screen "Configuraciones_3" 800x480, template "Template_3"
   IOField "I/O field_1" at 51,95 size 96x32; FormatPattern s99999
      ProcessValue <- "UDT_Objetos_Bombas_BC-11_frecuencia"
   TextField "Text field_1" at 75,36 size 32x20; Text 'XXX'
   TextField "Text field_3" at 60,57 size 74x36; Text 'Frecuencia Trabajo'
   IOField "I/O field_3" at 49,241 size 96x32; FormatPattern 999
      ProcessValue <- "UDT_Objetos_Sensores_Especiales_COT-01_operacion_bajo"
   TextField "Text field_4" at 71,180 size 32x20; Text 'XXX'
   TextField "Text field_5" at 40,202 size 114x36; Text 'Rango operación bajo'
   IOField "I/O field_4" at 49,314 size 96x32; FormatPattern 999
      ProcessValue <- "UDT_Objetos_Sensores_Especiales_COT-01_operacion_alto"
   TextField "Text field_6" at 40,275 size 114x36; Text 'Rango operación alto'
   IOField "I/O field_5" at 49,387 size 96x32; FormatPattern 999
      ProcessValue <- "UDT_Objetos_Sensores_Especiales_COT-01_trabajo_alto"
   TextField "Text field_7" at 63,348 size 67x36; Text 'Punto de trabajo'
   IOField "I/O field_6" at 201,240 size 96x32; FormatPattern 9999
      ProcessValue <- "UDT_Objetos_Flujo_FI-11_operacion_alto"
   TextField "Text field_8" at 295,179 size 38x20; Text 'FI-11'
   TextField "Text field_9" at 192,201 size 114x36; Text 'Rango operación bajo'
   IOField "I/O field_7" at 201,313 size 96x32; FormatPattern 9999
      ProcessValue <- "UDT_Objetos_Flujo_FI-11_operacion_alto"
   TextField "Text field_10" at 192,274 size 114x36; Text 'Rango operación alto'
   IOField "I/O field_8" at 201,386 size 96x32; FormatPattern 9999
      ProcessValue <- "UDT_Objetos_Flujo_FI-11_trabajo_alto"
   TextField "Text field_11" at 208,347 size 82x36; Text 'Punto de trabajo alto'
   IOField "I/O field_9" at 331,240 size 96x32; FormatPattern 9999
      ProcessValue <- "UDT_Objetos_Flujo_FI-11_trabajo_bajo"
   TextField "Text field_12" at 338,201 size 85x36; Text 'Punto de trabajo bajo'
   IOField "I/O field_2" at 484,240 size 96x32; FormatPattern s9999
      ProcessValue <- "UDT_Objetos_Flujo_FI-09_operacion_bajo"
   TextField "Text field_2" at 572,179 size 32x20; Text 'XXX'
   TextField "Text field_13" at 475,201 size 114x36; Text 'Rango operación bajo'
   IOField "I/O field_10" at 484,313 size 96x32; FormatPattern s9999
      ProcessValue <- "UDT_Objetos_Flujo_FI-09_operacion_alto"
   TextField "Text field_14" at 475,274 size 114x36; Text 'Rango operación alto'
   IOField "I/O field_11" at 484,386 size 96x32; FormatPattern s9999
      ProcessValue <- "UDT_Objetos_Flujo_FI-09_trabajo_alto"
   TextField "Text field_15" at 491,347 size 82x36; Text 'Punto de trabajo alto'
   IOField "I/O field_12" at 614,240 size 96x32; FormatPattern s9999
      ProcessValue <- "UDT_Objetos_Flujo_FI-09_trabajo_bajo"
   TextField "Text field_16" at 621,201 size 85x36; Text 'Punto de trabajo bajo'
   Button "Template_Button_7" at 0,440 size 99x39; TextOff 'COT'; PictureOff "Left_Arrow"
      on Click: ActivateScreen("Configuraciones_2", 0)
   Button "Template_Button_8" at 700,441 size 99x39; TextOff 'PT'; PictureOff "Right_Arrow"
      on Click: ActivateScreen("Configuraciones_4", 0)

screen "Configuraciones_4" 800x480, template "Template_3"
   IOField "I/O field_1" at 51,95 size 96x32; FormatPattern s99999
      ProcessValue <- "UDT_Objetos_Bombas_BC-11_frecuencia"
   TextField "Text field_1" at 75,36 size 32x20; Text 'XXX'
   TextField "Text field_3" at 60,57 size 74x36; Text 'Frecuencia Trabajo'
   IOField "I/O field_3" at 49,241 size 96x32; FormatPattern 999
      ProcessValue <- "UDT_Objetos_Sensores_Especiales_COT-01_operacion_bajo"
   TextField "Text field_4" at 71,180 size 32x20; Text 'XXX'
   TextField "Text field_5" at 40,202 size 114x36; Text 'Rango operación bajo'
   IOField "I/O field_4" at 49,314 size 96x32; FormatPattern 999
      ProcessValue <- "UDT_Objetos_Sensores_Especiales_COT-01_operacion_alto"
   TextField "Text field_6" at 40,275 size 114x36; Text 'Rango operación alto'
   IOField "I/O field_5" at 49,387 size 96x32; FormatPattern 999
      ProcessValue <- "UDT_Objetos_Sensores_Especiales_COT-01_trabajo_alto"
   TextField "Text field_7" at 63,348 size 67x36; Text 'Punto de trabajo'
   IOField "I/O field_6" at 201,240 size 96x32; FormatPattern 9999
      ProcessValue <- "UDT_Objetos_Flujo_FI-08_operacion_bajo"
   TextField "Text field_8" at 295,179 size 38x20; Text 'FI-08'
   TextField "Text field_9" at 192,201 size 114x36; Text 'Rango operación bajo'
   IOField "I/O field_7" at 201,313 size 96x32; FormatPattern 9999
      ProcessValue <- "UDT_Objetos_Flujo_FI-08_operacion_alto"
   TextField "Text field_10" at 192,274 size 114x36; Text 'Rango operación alto'
   IOField "I/O field_8" at 201,386 size 96x32; FormatPattern 9999
      ProcessValue <- "UDT_Objetos_Flujo_FI-08_trabajo_alto"
   TextField "Text field_11" at 208,347 size 82x36; Text 'Punto de trabajo alto'
   IOField "I/O field_9" at 331,240 size 96x32; FormatPattern 9999
      ProcessValue <- "UDT_Objetos_Flujo_FI-08_trabajo_bajo"
   TextField "Text field_12" at 338,201 size 85x36; Text 'Punto de trabajo bajo'
   IOField "I/O field_2" at 484,240 size 96x32; FormatPattern s9999
      ProcessValue <- "UDT_Objetos_Flujo_FI-09_operacion_bajo"
   TextField "Text field_2" at 572,179 size 38x20; Text 'FI-09'
   TextField "Text field_13" at 475,201 size 114x36; Text 'Rango operación bajo'
   IOField "I/O field_10" at 484,313 size 96x32; FormatPattern s9999
      ProcessValue <- "UDT_Objetos_Flujo_FI-09_operacion_alto"
   TextField "Text field_14" at 475,274 size 114x36; Text 'Rango operación alto'
   IOField "I/O field_11" at 484,386 size 96x32; FormatPattern s9999
      ProcessValue <- "UDT_Objetos_Flujo_FI-09_trabajo_alto"
   TextField "Text field_15" at 491,347 size 82x36; Text 'Punto de trabajo alto'
   IOField "I/O field_12" at 614,240 size 96x32; FormatPattern s9999
      ProcessValue <- "UDT_Objetos_Flujo_FI-09_trabajo_bajo"
   TextField "Text field_16" at 621,201 size 85x36; Text 'Punto de trabajo bajo'
   Button "Template_Button_7" at 0,440 size 99x39; TextOff 'COT'; PictureOff "Left_Arrow"
      on Click: ActivateScreen("Configuraciones_3", 0)
   Button "Template_Button_8" at 700,441 size 99x39; TextOff 'PT'; PictureOff "Right_Arrow"
      on Click: ActivateScreen("Configuraciones_5", 0)

screen "Configuraciones_5" 800x480, template "Template_3"
   IOField "I/O field_6" at 80,88 size 96x32; FormatPattern 9999; Unit  m
      ProcessValue <- "UDT_Objetos_Nivel_RAD-04_rango_alto"
   TextField "Text field_8" at 101,22 size 55x20; Text 'RAD-04'
   TextField "Text field_9" at 71,44 size 114x36; Text 'Rango operacion alto'
   IOField "I/O field_7" at 80,157 size 96x32; FormatPattern 9999; Unit  m
      ProcessValue <- "UDT_Objetos_Nivel_RAD-04_rango_bajo"
   TextField "Text field_10" at 95,129 size 67x20; Text 'Nivel bajo'
   IOField "I/O field_8" at 80,242 size 96x32; FormatPattern 9999; Unit  m
      ProcessValue <- "UDT_Objetos_Nivel_RAD-04_rango_medio_bajo"
   TextField "Text field_11" at 90,198 size 77x36; Text 'Nivel medio bajo'
   IOField "I/O field_9" at 80,327 size 96x32; FormatPattern 9999; Unit  m
      ProcessValue <- "UDT_Objetos_Nivel_RAD-04_rango_medio_alto"
   TextField "Text field_12" at 90,283 size 77x36; Text 'Nivel medio alto'
   IOField "I/O field_1" at 80,397 size 96x32; FormatPattern 9999; Unit  m
      ProcessValue <- "UDT_Objetos_Nivel_RAD-04_rango_alto"
   TextField "Text field_1" at 96,368 size 64x20; Text 'Nivel alto'
   IOField "I/O field_11" at 617,87 size 96x32; FormatPattern 9999; Unit  m
      ProcessValue <- "UDT_Objetos_Nivel_RAD-06_rango_alto"
   TextField "Text field_13" at 638,21 size 55x20; Text 'RAD-06'
   TextField "Text field_14" at 608,43 size 114x36; Text 'Rango operacion alto'
   IOField "I/O field_12" at 617,156 size 96x32; FormatPattern 9999; Unit  m
      ProcessValue <- "UDT_Objetos_Nivel_RAD-06_rango_bajo"
   TextField "Text field_15" at 632,128 size 67x20; Text 'Nivel bajo'
   IOField "I/O field_13" at 617,241 size 96x32; FormatPattern 9999; Unit  m
      ProcessValue <- "UDT_Objetos_Nivel_RAD-06_rango_medio_bajo"
   TextField "Text field_16" at 627,197 size 77x36; Text 'Nivel medio bajo'
   IOField "I/O field_14" at 617,326 size 96x32; FormatPattern 9999; Unit  m
      ProcessValue <- "UDT_Objetos_Nivel_RAD-06_rango_medio_alto"
   TextField "Text field_17" at 627,282 size 77x36; Text 'Nivel medio alto'
   IOField "I/O field_15" at 617,396 size 96x32; FormatPattern 9999; Unit  m
      ProcessValue <- "UDT_Objetos_Nivel_RAD-06_rango_alto(1)"
   TextField "Text field_18" at 633,367 size 64x20; Text 'Nivel alto'
   IOField "I/O field_2" at 350,88 size 96x32; FormatPattern 9999; Unit  m
      ProcessValue <- "UDT_Objetos_Nivel_RAD-05_rango_alto"
   TextField "Text field_2" at 371,22 size 55x20; Text 'RAD-05'
   TextField "Text field_3" at 341,44 size 114x36; Text 'Rango operacion alto'
   IOField "I/O field_3" at 350,157 size 96x32; FormatPattern 9999; Unit  m
      ProcessValue <- "UDT_Objetos_Nivel_RAD-05_rango_bajo"
   TextField "Text field_4" at 365,129 size 67x20; Text 'Nivel bajo'
   IOField "I/O field_4" at 350,242 size 96x32; FormatPattern 9999; Unit  m
      ProcessValue <- "UDT_Objetos_Nivel_RAD-05_rango_medio_bajo"
   TextField "Text field_5" at 360,198 size 77x36; Text 'Nivel medio bajo'
   IOField "I/O field_5" at 350,327 size 96x32; FormatPattern 9999; Unit  m
      ProcessValue <- "UDT_Objetos_Nivel_RAD-05_rango_medio_alto"
   TextField "Text field_6" at 360,283 size 77x36; Text 'Nivel medio alto'
   IOField "I/O field_10" at 350,397 size 96x32; FormatPattern 9999; Unit  m
      ProcessValue <- "UDT_Objetos_Nivel_RAD-05_rango_alto"
   TextField "Text field_7" at 366,368 size 64x20; Text 'Nivel alto'
   Button "Template_Button_7" at 0,440 size 99x39; TextOff 'COT'; PictureOff "Left_Arrow"
      on Click: ActivateScreen("Configuraciones_4", 0)
   Button "Template_Button_8" at 700,441 size 99x39; TextOff 'PT'; PictureOff "Right_Arrow"
      on Click: ActivateScreen("Presion", 0)

screen "Presion" 800x480, template "Template_3"
   IOField "I/O field_6" at 20,87 size 96x32; FormatPattern 9999; Unit  Bar
      ProcessValue <- "UDT_Objetos_Presion_PT-05_operacion_bajo"
   TextField "Text field_8" at 114,26 size 42x20; Text 'PT-05'
   TextField "Text field_9" at 11,48 size 114x36; Text 'Rango operación bajo'
   IOField "I/O field_7" at 20,160 size 96x32; FormatPattern 9999; Unit  Bar
      ProcessValue <- "UDT_Objetos_Presion_PT-05_operacion_alto"
   TextField "Text field_10" at 11,121 size 114x36; Text 'Rango operación alto'
   IOField "I/O field_8" at 149,160 size 96x32; FormatPattern 9999; Unit  Bar
      ProcessValue <- "UDT_Objetos_Presion_PT-05_trabajo_alto"
   TextField "Text field_11" at 156,121 size 82x36; Text 'Punto de trabajo alto'
   IOField "I/O field_9" at 150,87 size 96x32; FormatPattern 9999; Unit  Bar
      ProcessValue <- "UDT_Objetos_Presion_PT-05_trabajo_bajo"
   TextField "Text field_12" at 157,48 size 85x36; Text 'Punto de trabajo bajo'
   Group "Group" at 5,16 size 259x198
   IOField "I/O field_13" at 20,295 size 96x32; FormatPattern 9999; Unit  Bar
      ProcessValue <- "UDT_Objetos_Presion_PT-09_operacion_bajo"
   TextField "Text field_16" at 114,234 size 42x20; Text 'PT-09'
   TextField "Text field_17" at 11,256 size 114x36; Text 'Rango operación bajo'
   IOField "I/O field_14" at 20,368 size 96x32; FormatPattern 9999; Unit  Bar
      ProcessValue <- "UDT_Objetos_Presion_PT-09_operacion_alto"
   TextField "Text field_18" at 11,329 size 114x36; Text 'Rango operación alto'
   IOField "I/O field_15" at 149,368 size 96x32; FormatPattern 9999; Unit  Bar
      ProcessValue <- "UDT_Objetos_Presion_PT-09_trabajo_alto"
   TextField "Text field_19" at 156,329 size 82x36; Text 'Punto de trabajo alto'
   IOField "I/O field_16" at 150,295 size 96x32; FormatPattern 9999; Unit  Bar
      ProcessValue <- "UDT_Objetos_Presion_PT-09_trabajo_bajo"
   TextField "Text field_20" at 157,256 size 85x36; Text 'Punto de trabajo bajo'
   IOField "I/O field_17" at 286,295 size 96x32; FormatPattern 9999; Unit  Bar
      ProcessValue <- "UDT_Objetos_Presion_PT-10_operacion_bajo"
   TextField "Text field_21" at 380,234 size 42x20; Text 'PT-10'
   TextField "Text field_22" at 277,256 size 114x36; Text 'Rango operación bajo'
   IOField "I/O field_18" at 286,368 size 96x32; FormatPattern 9999; Unit  Bar
      ProcessValue <- "UDT_Objetos_Presion_PT-10_operacion_alto"
   TextField "Text field_23" at 277,329 size 114x36; Text 'Rango operación alto'
   IOField "I/O field_19" at 415,368 size 96x32; FormatPattern 9999; Unit  Bar
      ProcessValue <- "UDT_Objetos_Presion_PT-10_trabajo_alto"
   TextField "Text field_24" at 422,329 size 82x36; Text 'Punto de trabajo alto'
   IOField "I/O field_20" at 416,295 size 96x32; FormatPattern 9999; Unit  Bar
      ProcessValue <- "UDT_Objetos_Presion_PT-10_trabajo_bajo"
   TextField "Text field_25" at 423,256 size 85x36; Text 'Punto de trabajo bajo'
   IOField "I/O field_21" at 553,295 size 96x32; FormatPattern 9999; Unit  Bar
      ProcessValue <- "UDT_Objetos_Presion_PT-11_operacion_bajo"
   TextField "Text field_26" at 647,234 size 42x20; Text 'PT-11'
   TextField "Text field_27" at 544,256 size 114x36; Text 'Rango operación bajo'
   IOField "I/O field_22" at 553,368 size 96x32; FormatPattern 9999; Unit  Bar
      ProcessValue <- "UDT_Objetos_Presion_PT-11_operacion_alto"
   TextField "Text field_28" at 544,329 size 114x36; Text 'Rango operación alto'
   IOField "I/O field_23" at 682,368 size 96x32; FormatPattern 9999; Unit  Bar
      ProcessValue <- "UDT_Objetos_Presion_PT-11_trabajo_alto"
   TextField "Text field_29" at 689,329 size 82x36; Text 'Punto de trabajo alto'
   IOField "I/O field_24" at 683,295 size 96x32; FormatPattern 9999; Unit  Bar
      ProcessValue <- "UDT_Objetos_Presion_PT-11_trabajo_bajo"
   TextField "Text field_30" at 690,256 size 85x36; Text 'Punto de trabajo bajo'
   IOField "I/O field_1" at 286,87 size 96x32; FormatPattern 9999; Unit  Bar
      ProcessValue <- "UDT_Objetos_Presion_PT-06_operacion_bajo"
   TextField "Text field_1" at 380,26 size 42x20; Text 'PT-06'
   TextField "Text field_2" at 277,48 size 114x36; Text 'Rango operación bajo'
   IOField "I/O field_2" at 286,160 size 96x32; FormatPattern 9999; Unit  Bar
      ProcessValue <- "UDT_Objetos_Presion_PT-06_operacion_alto"
   TextField "Text field_3" at 277,121 size 114x36; Text 'Rango operación alto'
   IOField "I/O field_3" at 415,160 size 96x32; FormatPattern 9999; Unit  Bar
      ProcessValue <- "UDT_Objetos_Presion_PT-06_trabajo_alto"
   TextField "Text field_4" at 422,121 size 82x36; Text 'Punto de trabajo alto'
   IOField "I/O field_4" at 416,87 size 96x32; FormatPattern 9999; Unit  Bar
      ProcessValue <- "UDT_Objetos_Presion_PT-06_trabajo_bajo"
   TextField "Text field_5" at 423,48 size 85x36; Text 'Punto de trabajo bajo'
   IOField "I/O field_5" at 553,87 size 96x32; FormatPattern 9999; Unit  Bar
      ProcessValue <- "UDT_Objetos_Presion_PT-08_operacion_bajo"
   TextField "Text field_6" at 647,26 size 42x20; Text 'PT-08'
   TextField "Text field_7" at 544,48 size 114x36; Text 'Rango operación bajo'
   IOField "I/O field_10" at 553,160 size 96x32; FormatPattern 9999; Unit  Bar
      ProcessValue <- "UDT_Objetos_Presion_PT-08_operacion_alto"
   TextField "Text field_13" at 544,121 size 114x36; Text 'Rango operación alto'
   IOField "I/O field_11" at 682,160 size 96x32; FormatPattern 9999; Unit  Bar
      ProcessValue <- "UDT_Objetos_Presion_PT-08_trabajo_alto"
   TextField "Text field_14" at 689,121 size 82x36; Text 'Punto de trabajo alto'
   IOField "I/O field_12" at 683,87 size 96x32; FormatPattern 9999; Unit  Bar
      ProcessValue <- "UDT_Objetos_Presion_PT-08_trabajo_bajo"
   TextField "Text field_15" at 690,48 size 85x36; Text 'Punto de trabajo bajo'
   Button "Template_Button_7" at 0,440 size 99x39; TextOff 'COT'; PictureOff "Left_Arrow"
      on Click: ActivateScreen("Configuraciones_5", 0)
   Button "Template_Button_8" at 700,441 size 99x39; TextOff 'PT'; PictureOff "Right_Arrow"
      on Click: ActivateScreen("Presion2", 0)

screen "Presion2" 800x480, template "Template_3"
   IOField "I/O field_6" at 80,88 size 96x32; FormatPattern 9999; Unit  m
      ProcessValue <- "UDT_Objetos_Nivel_PT-07_operacion_alto"
   TextField "Text field_8" at 101,22 size 42x20; Text 'PT-07'
   TextField "Text field_9" at 71,44 size 114x36; Text 'Rango operacion alto'
   IOField "I/O field_7" at 80,157 size 96x32; FormatPattern 9999; Unit  m
      ProcessValue <- "UDT_Objetos_Nivel_PT-07_rango_bajo"
   TextField "Text field_10" at 95,129 size 67x20; Text 'Nivel bajo'
   IOField "I/O field_8" at 80,242 size 96x32; FormatPattern 9999; Unit  m
      ProcessValue <- "UDT_Objetos_Nivel_PT-07_rango_medio_bajo"
   TextField "Text field_11" at 90,198 size 77x36; Text 'Nivel medio bajo'
   IOField "I/O field_9" at 80,327 size 96x32; FormatPattern 9999; Unit  m
      ProcessValue <- "UDT_Objetos_Nivel_PT-07_rango_medio_alto"
   TextField "Text field_12" at 90,283 size 77x36; Text 'Nivel medio alto'
   IOField "I/O field_1" at 80,397 size 96x32; FormatPattern 9999; Unit  m
      ProcessValue <- "UDT_Objetos_Nivel_PT-07_rango_alto"
   TextField "Text field_1" at 96,368 size 64x20; Text 'Nivel alto'
   IOField "I/O field_11" at 617,87 size 96x32; FormatPattern 9999; Unit  m
      ProcessValue <- "UDT_Objetos_Nivel_PT-13_operacion_alto"
   TextField "Text field_13" at 638,21 size 42x20; Text 'PT-13'
   TextField "Text field_14" at 608,43 size 114x36; Text 'Rango operacion alto'
   IOField "I/O field_12" at 617,156 size 96x32; FormatPattern 9999; Unit  m
      ProcessValue <- "UDT_Objetos_Nivel_PT-13_rango_bajo"
   TextField "Text field_15" at 632,128 size 67x20; Text 'Nivel bajo'
   IOField "I/O field_13" at 617,241 size 96x32; FormatPattern 9999; Unit  m
      ProcessValue <- "UDT_Objetos_Nivel_PT-13_rango_medio_bajo"
   TextField "Text field_16" at 627,197 size 77x36; Text 'Nivel medio bajo'
   IOField "I/O field_14" at 617,326 size 96x32; FormatPattern 9999; Unit  m
      ProcessValue <- "UDT_Objetos_Nivel_PT-13_rango_medio_alto"
   TextField "Text field_17" at 627,282 size 77x36; Text 'Nivel medio alto'
   IOField "I/O field_15" at 617,396 size 96x32; FormatPattern 9999; Unit  m
      ProcessValue <- "UDT_Objetos_Nivel_PT-13_rango_alto"
   TextField "Text field_18" at 633,367 size 64x20; Text 'Nivel alto'
   IOField "I/O field_2" at 350,88 size 96x32; FormatPattern 9999; Unit  m
      ProcessValue <- "UDT_Objetos_Nivel_PT-12_operacion_alto"
   TextField "Text field_2" at 371,22 size 42x20; Text 'PT-12'
   TextField "Text field_3" at 341,44 size 114x36; Text 'Rango operacion alto'
   IOField "I/O field_3" at 350,157 size 96x32; FormatPattern 9999; Unit  m
      ProcessValue <- "UDT_Objetos_Nivel_PT-12_rango_bajo"
   TextField "Text field_4" at 365,129 size 67x20; Text 'Nivel bajo'
   IOField "I/O field_4" at 350,242 size 96x32; FormatPattern 9999; Unit  m
      ProcessValue <- "UDT_Objetos_Nivel_PT-12_rango_medio_bajo"
   TextField "Text field_5" at 360,198 size 77x36; Text 'Nivel medio bajo'
   IOField "I/O field_5" at 350,327 size 96x32; FormatPattern 9999; Unit  m
      ProcessValue <- "UDT_Objetos_Nivel_PT-12_rango_medio_alto"
   TextField "Text field_6" at 360,283 size 77x36; Text 'Nivel medio alto'
   IOField "I/O field_10" at 350,397 size 96x32; FormatPattern 9999; Unit  m
      ProcessValue <- "UDT_Objetos_Nivel_PT-12_rango_alto"
   TextField "Text field_7" at 366,368 size 64x20; Text 'Nivel alto'
   Button "Template_Button_7" at 0,440 size 99x39; TextOff 'COT'; PictureOff "Left_Arrow"
      on Click: ActivateScreen("COT", 0)
   Button "Template_Button_8" at 700,441 size 99x39; TextOff 'PT'; PictureOff "Right_Arrow"
      on Click: ActivateScreen("PT", 0)

screen "COT" 800x480, template "Template_2"
   TrendView "Trend view_1" at 0,57 size 800x383

screen "Produccion UF" 800x480, template "Alarmas"
   Button "Button_1" at 23,130 size 106x56; TextOff 'START'
   Button "Button_2" at 23,199 size 106x56; TextOff 'STOP'
   TextField "Text field_1" at 306,45 size 184x34; Text 'Producción UF'

screen "CT" 800x480, template "Template_2"
   TrendView "Trend view_1" at 0,57 size 800x383

screen "ORP" 800x480, template "Template_2"
   TrendView "Trend view_1" at 0,57 size 800x383

screen "PH" 800x480, template "Template_2"
   TrendView "Trend view_1" at 0,57 size 800x383

screen "TRB" 800x480, template "Template_2"
   TrendView "Trend view_1" at 0,57 size 800x383

screen "FI" 800x480, template "Template_2"
   TrendView "Trend view_1" at 0,57 size 800x383
   Button "Template_Button_7" at 699,0 size 99x39; TextOff 'FLUJO 2'
      on Click: ActivateScreen("COT", 0)

screen "RAD" 800x480, template "Template_2"
   TrendView "Trend view_1" at 0,57 size 800x383
   Button "Template_Button_7" at 699,0 size 99x39; TextOff 'NIVEL 1'
      on Click: ActivateScreen("COT", 0)

screen "PT" 800x480, template "Template_2"
   TrendView "Trend view_1" at 0,57 size 800x383
   Button "Template_Button_7" at 699,0 size 99x39; TextOff 'PRESION 2'
      on Click: ActivateScreen("COT", 0)

screen "FI_1" 800x480, template "Template_2"
   TrendView "Trend view_1" at 0,57 size 800x383
   Button "Template_Button_7" at 699,0 size 99x39; TextOff 'FLUJO 1'
      on Click: ActivateScreen("COT", 0)

screen "PT_1" 800x480, template "Template_2"
   TrendView "Trend view_1" at 0,57 size 800x383
   Button "Template_Button_7" at 699,0 size 99x39; TextOff 'PRESION 2'
      on Click: ActivateScreen("COT", 0)

screen "RAD_1" 800x480, template "Template_2"
   TrendView "Trend view_1" at 0,57 size 800x383
   Button "Template_Button_7" at 699,0 size 99x39; TextOff 'NIVEL 2'
      on Click: ActivateScreen("COT", 0)

screen "Alarmas" 800x480, template "Alarmas"
   AlarmView "Alarm view_1" at 8,8 size 785x382

Template "Template_3" 800x480
   Button "Template_Button_9" at 96,440 size 99x39; TextOff 'INICIO'
      on Click: ActivateScreen("0Ultrafiltracion", 0)

screen "Produccion OI" 800x480, template "Alarmas"
   Button "Button_1" at 23,130 size 106x56; TextOff 'START'
   Button "Button_2" at 23,199 size 106x56; TextOff 'STOP'
   TextField "Text field_1" at 306,45 size 182x34; Text 'Producción OI'

screen "Produccion PER" 800x480, template "Alarmas"
   Button "Button_1" at 23,130 size 106x56; TextOff 'START'
   Button "Button_2" at 23,199 size 106x56; TextOff 'STOP'
   TextField "Text field_1" at 306,45 size 200x34; Text 'Producción PER'

Template "Alarmas" 800x480
   Button "Template_Button_3" at 400,440 size 100x39; TextOff 'MANUAL'
      on Click: ActivateScreen("Manual", 0)
   Button "Template_Button_4" at 300,440 size 100x39; TextOff 'GRAFICAS'
      on Click: ActivateScreen("COT", 0)
   Button "Template_Button_5" at 200,440 size 100x39; TextOff 'PRODUCCION PER'
      on Click: ActivateScreen("Produccion PER", 0)
   Button "Template_Button_6" at 100,440 size 100x39; TextOff 'PRODUCCION OI'
      on Click: ActivateScreen("Produccion OI", 0)
   Button "Template_Button_7" at 0,440 size 100x39; TextOff 'PRODUCCION UF'
      on Click: ActivateScreen("Produccion UF", 0)
   Button "Template_Button_9" at 500,440 size 99x39; TextOff 'INICIO'
      on Click: ActivateScreen("0Ultrafiltracion", 0)

screen "Proceso UF" 800x480, template "Template_3"
   IOField "I/O field_6" at 80,88 size 96x32; FormatPattern 9999; Unit  m
      ProcessValue <- "UDT_Objetos_Nivel_PT-07_operacion_alto"
   TextField "Text field_8" at 379,22 size 42x20; Text 'PT-07'
   TextField "Text field_9" at 71,44 size 114x36; Text 'Rango operacion alto'
   IOField "I/O field_7" at 80,157 size 96x32; FormatPattern 9999; Unit  m
      ProcessValue <- "UDT_Objetos_Nivel_PT-07_rango_bajo"
   TextField "Text field_10" at 95,129 size 67x20; Text 'Nivel bajo'
   IOField "I/O field_8" at 80,242 size 96x32; FormatPattern 9999; Unit  m
      ProcessValue <- "UDT_Objetos_Nivel_PT-07_rango_medio_bajo"
   TextField "Text field_11" at 90,198 size 77x36; Text 'Nivel medio bajo'
   IOField "I/O field_9" at 80,327 size 96x32; FormatPattern 9999; Unit  m
      ProcessValue <- "UDT_Objetos_Nivel_PT-07_rango_medio_alto"
   TextField "Text field_12" at 90,283 size 77x36; Text 'Nivel medio alto'
   IOField "I/O field_1" at 80,397 size 96x32; FormatPattern 9999; Unit  m
      ProcessValue <- "UDT_Objetos_Nivel_PT-07_rango_alto"
   TextField "Text field_1" at 96,368 size 64x20; Text 'Nivel alto'
   Button "Template_Button_7" at 0,440 size 99x39; TextOff 'COT'; PictureOff "Left_Arrow"
      on Click: ActivateScreen("COT", 0)
   Button "Template_Button_8" at 700,441 size 99x39; TextOff 'PT'; PictureOff "Right_Arrow"
      on Click: ActivateScreen("PT", 0)
*)